{attribute 'qualified_only'}
{attribute 'strict'}
TYPE eLogTypes :
(
	TrackCycles := 0,
	TrackOnTime	:= 1,
	WriteValue := 2,
	KeepHighestValue := 3,
	KeepLowestValue	:= 4
);
END_TYPE

(* stored: Version 1.1.0.1, ProductVersion 3.1.4026.18
   DUT eLogTypes: Id {8db96618-bfd9-49a0-bfd3-740e573c33ff} *)
